FUNCTION_BLOCK PUBLIC FB_PositionTrigger_Old // trigger function, sets trigger Q signal high when trigger position is between previous cycle's and current axis position.
VAR_INPUT
	fAxisPos			: LREAL	; // Axis position on which the to trigger
	nAxisModuloRev		: DINT 	:= 0	; // axis modulo revolutions 
	fAxisVelocity		: LREAL := 0 	; 	// velocity of axis 
	bDirPositive		: BOOL 	:= TRUE ; // Axis direction is forward 
	fEncoderTurnover	: LREAL	:= 360 	; // Encoder turnover value (standard 360 deg)
	bEnablenNegative 	: BOOL 	:= FALSE; // Enables negative input values
END_VAR
VAR_OUTPUT
	Q					: BOOL 	; // trigger signal
	bInternalTrigger	: BOOL 	; // Internal trigger signal 
	bTriggerArmed 		: BOOL 	; // Trigger is armed 
	bEncoderTurnedOver	: BOOL 	; // is high when encoder goes thru it's turnover point 
	fAccuracy 			: LREAL ; // Accuracy of trigger 
END_VAR
VAR
	// function commands
	fTriggerPosition 		: LREAL ; // trigger position 
	fTriggerPosCompensated	: LREAL ; // TRigger Position after compensation
	nRotBeforeTrigger		: DINT 	:= 0 ; 	// Full axis rotations before position trigger is armed
	nRotBeforeTriggerCompensated	: DINT := 0 ; // full E_ComponentTypes.Axis rotation before trigger IsFinite armed 
	// Trigger variables 
	fReactionTime			: LREAL	:= 0 ; 	// [ms] Time before reaction to trigger (time compensation)
	// internal values	
	nTriggerRotation		: DINT	:= 0 ; 	// Number of rotations done since trigger is armed 
	fOldAxisPos				: LREAL ; 		// Old axis position for comparison
	nOldAxisRev				: DINT 	; 		// Old modulo revolutions 
	fCompensationDistance	: LREAL := 0 ; 	// [units] trigger compensation distance  
	// Edge functions 
	fbReTriggerArmed		: R_TRIG ; // rising edge trigger on trigger armed (used to rest trigger values) 
END_VAR

// Rising edge function execute
fbReTriggerArmed(CLK := bTriggerArmed); 

// ==== Skip function if trigger is not armed =====
	IF NOT bTriggerArmed THEN  
		bInternalTrigger	:= FALSE 	;
		Q 					:= FALSE	;
		RETURN ;	
	ELSIF fbReTriggerArmed.Q THEN 
		fOldAxisPos 		:= fAxisPos ;
		nOldAxisRev			:= nAxisModuloRev ;
		nTriggerRotation	:= 0 		; 
	END_IF
	
// ==== check if encoder is at turnover =====
	ExecTurnoverCheck(); 
// ==== compare positions to trigger ======
	CalcTriggerCompensation();
	ExecArmTrigger();

METHOD PRIVATE CalcTriggerCompensation : BOOL
VAR_INPUT
END_VAR
// ===== Calculate the distance travelled within the delay time =====
	fCompensationDistance	:= fReactionTime  * (fAxisVelocity / 1000);
END_METHOD

METHOD PUBLIC CmdArmTrigger : BOOL // arm trigger
VAR_INPUT
END_VAR
// Arm trigger command 
bTriggerArmed S= TRUE ;

// set feedback
CmdArmTrigger := NOT Q ;
END_METHOD

METHOD PUBLIC CmdSetTriggerPos : BOOL
VAR_INPUT
	fCmdPosition 	: LREAL ; // Trigger position 
	nCmdRotations	: DINT	:= 0 ; // Rotations before trigger is set  
	nCmdReactionTime: LREAL := 0 ; // [ms]reaction time to trigger signal 
END_VAR
// set trigger position
fTriggerPosition 	:= fCmdPosition ;
nRotBeforeTrigger	:= nCmdRotations;
fReactionTime 		:= nCmdReactionTime ;
END_METHOD

METHOD INTERNAL ExecArmTrigger : BOOL
VAR_INPUT
END_VAR
// ===== Retract compensationdistance from trigger distance =====

// check if trigger pos is not negative 
IF NOT bEnablenNegative AND fTriggerPosCompensated < 0 THEN
	fTriggerPosCompensated 			:= fEncoderTurnover + fTriggerPosition ;
	nRotBeforeTriggerCompensated	:= nRotBeforeTrigger -	1;  
ELSE
	fTriggerPosCompensated 			:= fTriggerPosition - fCompensationDistance ;
	nRotBeforeTriggerCompensated	:= nRotBeforeTrigger ;  
END_IF 

// ==== compare positions to trigger ======
	bInternalTrigger := FALSE ;

	IF bEncoderTurnedOver THEN
		IF bDirPositive THEN
			bInternalTrigger S= Between(fOldAxisPos , fTriggerPosCompensated, fEncoderTurnover) ;
			bInternalTrigger S= Between(0	, fTriggerPosCompensated, fAxisPos) ;
		ELSE 
			bInternalTrigger S= Between(0			, fTriggerPosCompensated, fOldAxisPos) ;
			bInternalTrigger S= Between(fAxisPos	, fTriggerPosCompensated, fEncoderTurnover) ;
		END_IF 
		bEncoderTurnedOver := FALSE ;
	ELSE 
		bInternalTrigger S= Between(fAxisPos	, fTriggerPosCompensated, fOldAxisPos) ;
		bInternalTrigger S= Between(fOldAxisPos	, fTriggerPosCompensated, fAxisPos) ;
		fAccuracy	:= ABS( fOldAxisPos - fAxisPos);
	END_IF

	fOldAxisPos := fAxisPos ;

// ==== Check multiturn command =======
	IF bInternalTrigger THEN 
		IF nTriggerRotation >= nRotBeforeTriggerCompensated THEN 
			Q S= bInternalTrigger OR fAxisPos > fTriggerPosCompensated;			
		ELSE 
			nTriggerRotation := nTriggerRotation + 1 ;
		END_IF 
	END_IF

// ==== Reset arm trigger command =====
	bTriggerArmed 	R= Q ;
END_METHOD

METHOD PRIVATE ExecTurnoverCheck : BOOL
VAR_INPUT
END_VAR
	bEncoderTurnedOver := nOldAxisRev <> nAxisModuloRev ;
	nOldAxisRev := nAxisModuloRev ;
END_METHOD

END_FUNCTION_BLOCK

(* stored: Version 1.1.0.1, ProductVersion 3.1.4024.5
   POU FB_PositionTrigger_Old: Id {fd987587-b4d1-405a-9d23-bb003d45ecc7}, SpecialFunc None
   Folder Private: Id {4208ffc7-0704-4b5d-8914-d67f25180c1c}
   Method CalcTriggerCompensation: Id {96ec8b32-d310-4326-901c-edd47b255ebf}
   Method CmdArmTrigger: Id {05a97c0b-39d0-42ba-8875-9046cdb77eac}
   Method CmdSetTriggerPos: Id {456097cb-6b4e-4349-a84a-cae4874abe8e}
   Method ExecArmTrigger: Id {53cf7f82-8ace-4dd1-a2b0-26e0d90c74fe}
   Method ExecTurnoverCheck: Id {10051210-68d4-4637-9383-f379a08b872f} *)
